FUNCTION_BLOCK HomeSequence
VAR_INPUT
	EN :BOOL;
	iHomeCycleStart :BOOL;
	iClampOpenGroup1 :BOOL;
	iClampOpenGroup2 :BOOL;
	iTT_at_0 : BOOL;
	iTrunion_at_0 :BOOL;
	iDoor_Cls : BOOL;
END_VAR
VAR_OUTPUT
	ENO :BOOL;
	qGroup1ClampOpen :BOOL;
	qGroup2ClampOpen :BOOL;
	qTT_0 : BOOL;
	qTrunion_0 : BOOL;
	qDoor_Cls : BOOL;
	qHomeDone : BOOL;
END_VAR
VAR
	StepNo : INT;
END_VAR

CASE StepNo OF
	
0:
	qHomeDone := FALSE;
	IF iHomeCycleStart THEN
	StepNo := 10;
	END_IF

// All Clamps home
10:
	qGroup1ClampOpen := TRUE;
	qGroup2ClampOpen := TRUE;
	IF iClampOpenGroup1 AND iClampOpenGroup2 THEN
		qGroup1ClampOpen := FALSE;
		qGroup2ClampOpen := FALSE;
		StepNo := 20;
	END_IF

// Roller door close
20:
	qDoor_Cls := TRUE;
	IF iDoor_Cls THEN
		qDoor_Cls := FALSE;
		StepNo := 30;
	END_IF
	
// Trunion to 0* position
30:
	qTrunion_0 := TRUE;
	IF iTrunion_at_0 THEN
		qTrunion_0 := FALSE;
		StepNo := 40;
	END_IF

// Turn Table to home position
40:
	qTT_0 := TRUE;
	IF iTT_at_0 THEN
		qTT_0 := FALSE;
		qHomeDone := TRUE;
		StepNo := 0;
	END_IF
	
END_CASE

END_FUNCTION_BLOCK

(* stored: Version 1.1.0.1, ProductVersion 3.1.4024.16
   POU HomeSequence: Id {5a6a5d55-439f-4a7f-955c-8529d4bdf1aa}, SpecialFunc None *)
